// TIA Portal V20 export
TYPE "zm_MachineMode"
// stored: Access Published
   STRUCT
      Manual : Bool;
      Auto : Bool;
      Maintenance : Bool;
      Nomode : Bool;
   END_STRUCT;
END_TYPE
